Staubli VAL3: stop.pgx

program stop()
begin
  // Se finaliza la aplicacion

  // Nada que hacer aqui!
end
